{attribute addProperty BoxType "EK1122-0000-0018"}
{attribute addProperty Id "Beckhoff_ER6xxxsub_EK1100EK1100_179A0949162A_0001_ER6001_0002_0016ER6001_4599C92248060A_0002_ER6001_0002_0021ER6001_4599C92248060A_0003_ER6002_0002_0021ER6002_6961C256864108A_0004_ER6002_0002_0022ER6002_E45E7FFD864108A_0005_ER6002_0002_0023ER6002_E45E7FFD864108"}
{attribute addProperty CRC "1866957675"}
{attribute addProperty SizeInBites "3568"}
{attribute addProperty SizeInBytes "446"}
TYPE Beckhoff_ER6xxxEK1122_6F47836B EXTENDS EK1122_179A0949 :
STRUCT
	{attribute addProperty Name "Beckhoff_ER6xxxsub_EK1100"}
	Beckhoff_ER6xxxsub_EK1100 : EK1100_179A0949;
	{attribute addProperty Name "A_0001_ER6001_0002_0016"}
	A_0001_ER6001_0002_0016 : ER6001_4599C922;
	{attribute addProperty Name "A_0002_ER6001_0002_0021"}
	A_0002_ER6001_0002_0021 : ER6001_4599C922;
	{attribute addProperty Name "A_0003_ER6002_0002_0021"}
	A_0003_ER6002_0002_0021 : ER6002_6961C256;
	{attribute addProperty Name "A_0004_ER6002_0002_0022"}
	A_0004_ER6002_0002_0022 : ER6002_E45E7FFD;
	{attribute addProperty Name "A_0005_ER6002_0002_0023"}
	A_0005_ER6002_0002_0023 : ER6002_E45E7FFD;
END_STRUCT
END_TYPE

(* stored: Version 1.2.0.0, ProductVersion 3.1.4024.9
   DUT Beckhoff_ER6xxxEK1122_6F47836B: Id {1dfacf4d-5dad-456e-9ab3-8870c657c123} *)
